{attribute 'GeneratedUsingTerminal: DL-EC1A-0000'}
{attribute addProperty BoxType "DL-EC1A-0000"}
{attribute addProperty Id "Error_StatusAT %I*BOOL1Error_CodeAT %I*UINT2"}
{attribute addProperty CRC "3460174704"}
{attribute addProperty Size "3"}
TYPE Status_of_System_CE3E1370 EXTENDS InputBase_8311D824 :
STRUCT
	{attribute addProperty Name "Error_Status"}
	Error_Status AT %I* : BOOL;
	{attribute addProperty Name "Error_Code"}
	Error_Code AT %I* : UINT;
END_STRUCT
END_TYPE
